// TwinCAT 3 PLC project Untitled1
// ProgramVersion: 3.1.4024.0
// libraries:
//   Tc2_Standard, * (Beckhoff Automation GmbH)
//   Tc2_System, * (Beckhoff Automation GmbH)
//   Tc3_IotCommunicator, * (Beckhoff Automation GmbH)
//   Tc3_Module, * (Beckhoff Automation GmbH)
// project tree:
//   DUTs/Floor 1/Lighting/ ST_Lighting.TcDUT, ST_LightingTemplate.TcDUT
//   DUTs/Floor 1/ ST_FloorOne.TcDUT, ST_RoomOne.TcDUT
//   GVLs/ House.TcGVL
//   / PlcTask.TcTTO
//   POUs/ Constants.TcPOU, MAIN.TcPOU
// real-time tasks:
//   TASK PlcTask: cycle T#10ms, priority 20, ADS port 350

CONFIGURATION Untitled1
    RESOURCE PLC ON TwinCAT3
        TASK PlcTask(INTERVAL := T#10ms, PRIORITY := 20);
        PROGRAM MAIN WITH PlcTask : MAIN;
    END_RESOURCE
END_CONFIGURATION

// ---- DUTs/Floor 1/Lighting/ST_Lighting.TcDUT
TYPE ST_Lighting :
STRUCT
	
	{attribute 'iot.ReadOnly' := 'false'}
	{attribute 'iot.DisplayName' := 'Floor Lighting'}
	{attribute 'iot.WidgetType' := 'Lighting'}
	{attribute 'iot.LightValueVisible' := 'false'}
	{attribute 'iot.LightSliderVisible' := 'true'}
	{attribute 'iot.LightModeVisible' := 'true'}
	{attribute 'iot.LightModeChangeable' := 'true'}
	stLighting	: ST_LightingTemplate;
	
END_STRUCT
END_TYPE

// ---- DUTs/Floor 1/Lighting/ST_LightingTemplate.TcDUT
TYPE ST_LightingTemplate :
STRUCT
	bLight		: BOOL;
	{attribute 'iot.Unit':='%'}
	{attribute 'iot.MinValue':='0'}
	{attribute 'iot.MaxValue':='100'}
	nLight		: INT;	
	sMode		: STRING ;
	aModes		: ARRAY[0..1] OF STRING;
END_STRUCT
END_TYPE

// ---- DUTs/Floor 1/ST_FloorOne.TcDUT
TYPE ST_FloorOne :
STRUCT
	
	{attribute 'iot.NestedStructIcon' := 'Lightbulb'}
	{attribute 'iot.DisplayName' := 'Light Widgets'}
	stLights		: ST_Lighting;
	
	{attribute 'iot.NestedStructIcon' := 'Room'}
	{attribute 'iot.DisplayName' := 'Confrence Room'}
	stRoomOne		: ST_RoomOne;

END_STRUCT
END_TYPE

// ---- DUTs/Floor 1/ST_RoomOne.TcDUT
TYPE ST_RoomOne :
STRUCT
	
	{attribute 'iot.DisplayName' := 'Projector'}
	 Projector : BOOL;
	 
	 
	 {attribute 'iot.NestedStructIcon' := 'Temperature'}
	 {attribute 'iot.Unit' := 'F'}
	 {attribute 'iot.DisplayName' := 'Temperature'}
	 {attribute 'iot.DecimalPrecision' := '2'}
	 {attribute 'iot.MinValue' := '60'} {attribute 'iot.MaxValue' := '90'}
	 {attribute 'iot.ReadOnly' := 'TRUE'}
	 ConTemp : LREAL := 75.2; 

END_STRUCT
END_TYPE

// ---- GVLs/House.TcGVL
{attribute 'qualified_only'}
VAR_GLOBAL
		stFloorOne	: ST_FloorOne;
END_VAR

// ---- POUs/MAIN.TcPOU
PROGRAM MAIN
VAR
	
	// Declare FB_IotCommunicator
	fbIot : FB_IotCommunicator := (sHostName := 'iot.beckhoff.us',
									nPort := 1883,
									sMainTopic := 'Test',
									sDeviceName := 'Automated Building',
									sDeviceIcon := 'House');
	
	// Timer to send data only once per second
	timer : TON;
	
	
	

END_VAR

// .Execute() has to be called cyclically
fbIot.Execute(TRUE);

// Start timer when fbIot is connected
IF fbIot.bConnected THEN
	timer(IN := TRUE, PT := T#500MS);
END_IF


// Send data, if timer is expired
IF timer.Q THEN
	timer(IN := FALSE);
	fbIot.SendData(ADR(House.stFloorOne), SIZEOF(House.stFloorOne));
END_IF



Lighting(); 
Constants();
Room_One();

METHOD Lighting 
VAR_INPUT
END_VAR
IF fbIot.fbCommand.bAvailable THEN
	// Receive data for first level struct

	IF fbIot.fbCommand.sVarName = 'stLights.stLighting.bLight' THEN
		fbIot.fbCommand.GetValue(ADR(House.stFloorOne.stLights.stLighting.bLight), SIZEOF(House.stFloorOne.stLights.stLighting.bLight), E_IotCommunicatorDatatype.type_BOOL);
	ELSIF fbIot.fbCommand.sVarName = 'stLights.stLighting.nLight' THEN
		fbIot.fbCommand.GetValue(ADR(House.stFloorOne.stLights.stLighting.nLight), SIZEOF(House.stFloorOne.stLights.stLighting.nLight), E_IotCommunicatorDatatype.type_INT);
	ELSIF fbIot.fbCommand.sVarName = 'stLights.stLighting.sMode' THEN
		fbIot.fbCommand.GetValue(ADR(House.stFloorOne.stLights.stLighting.sMode), SIZEOF(House.stFloorOne.stLights.stLighting.sMode), E_IotCommunicatorDatatype.type_STRING);
	END_IF
	fbIot.SendData(ADR(House.stFloorOne), SIZEOF(House.stFloorOne));
	fbIot.fbCommand.Remove();
END_IF

//Lighting Sample 2
House.stFloorOne.stLights.stLighting.aModes[0]:='Automatic';
House.stFloorOne.stLights.stLighting.aModes[1]:='Manual';
END_METHOD

METHOD Room_One 
VAR_INPUT
END_VAR
IF fbIot.fbCommand.bAvailable THEN
	// Receive data for first level struct

	IF fbIot.fbCommand.sVarName = 'stRoomOne.Projector' THEN
		fbIot.fbCommand.GetValue(ADR(House.stFloorOne.stRoomOne.Projector), SIZEOF(House.stFloorOne.stRoomOne.Projector), E_IotCommunicatorDatatype.type_BOOL);
	END_IF
	
	IF fbIot.fbCommand.sVarName = 'stRoomOne.ConTemp' THEN
		fbIot.fbCommand.GetValue(ADR(House.stFloorOne.stRoomOne.ConTemp), SIZEOF(House.stFloorOne.stRoomOne.ConTemp), E_IotCommunicatorDatatype.type_LREAL);
	END_IF
	
	fbIot.SendData(ADR(House.stFloorOne), SIZEOF(House.stFloorOne));
	fbIot.fbCommand.Remove();
END_IF
END_METHOD

END_PROGRAM

// ---- POUs/Constants.TcPOU
PROGRAM Constants
VAR
	
	bInit:BOOL:=TRUE;

END_VAR

IF bInit THEN
	bInit:=FALSE;
	//Lighting Init
	House.stFloorOne.stLights.stLighting.aModes[0]:='Automatic';
	House.stFloorOne.stLights.stLighting.aModes[1]:='Manual';
	House.stFloorOne.stLights.stLighting.sMode:='Init';
END_IF

END_PROGRAM
